SUBAPPLICATION SoftKey_Abscheider_UP (* Subapplication Type *)
  (* Standard: 61499-2 *)
  (* Version 1.0, 2023-02-06, franz *)
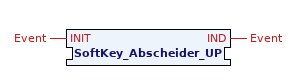
  EVENT_INPUT
    INIT;
  END_EVENT
  EVENT_OUTPUT
    IND;
  END_EVENT
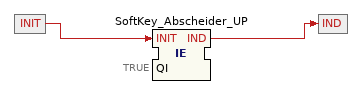
  FBS
    SoftKey_Abscheider_UP : IE(QI := TRUE);
  END_FBS
  EVENT_CONNECTIONS
    INIT TO SoftKey_Abscheider_UP.INIT;
    SoftKey_Abscheider_UP.IND TO IND;
  END_CONNECTIONS
END_SUBAPPLICATION
